Staubli VAL3: usrButtonTxt.pgx

program usrButtonTxt(num x_nWhichButton (dimensions=1), string x_sButtonTxt (dimensions=1))
begin
  //-----------------------------------------------------------------------
  //Header begin
  //Description of program
  //  This program lets you choose the button to display
  //
  //Input parameters
  //  num x_nWhichButton :
  //    role : choice of the navigation key
  //    possible values : 1 to 8 (F1 to F8)
  //
  //  string x_sButtonTxt :
  //    role : Displays desired text
  //
  //Traceability
  //  Creation : 07-04-08 - f.Rob
  //Header end
  //-----------------------------------------------------------------------

  //Position cursor X, Y
  gotoxy(nXPosButTxt[x_nWhichButton],nYPosButTxt)
  //Displays Text
  put(left(x_sButtonTxt,4))
  //Erases contents of  text button parameters
  x_sButtonTxt=" "
end
